Staubli VAL3: SYNCMOVE.pgx

public program syncMove(num& x_nAxisNum[])
  local jointRx l_jCurr
  local num l_nEncRes
  local num l_nDrvPos[2]
  local bool l_bFirstRun
  local num l_i
  local bool l_bError
  local string l_sMsg
begin

  l_nEncRes=8192/360

  call setCmdPos(0)
  call setCmdPos(1)
  bStop=false
  l_bFirstRun=true

  // Ne pas supprimer ces lignes
  disablePower()
  wait(isPowered()==false)
  //wait(isPowered()==true)
  /// FIN /////////////

  while !bStop
    if (isPowered()==true) and (l_bFirstRun==false)
      for l_i=0 to size(x_nAxisNum)-1
        if (diSwitchedOn[x_nAxisNum[l_i]]==false)
          doSwitchOn[x_nAxisNum[l_i]]=true
          delay(0.05)
          doEnableOp[x_nAxisNum[l_i]]=true
        endIf
      endFor
      // Get system position
      $XgetDrvCmdPos(l_nDrvPos)
      //$XgetJntCmdPos(l_nJntPos)
      // Send it to the external axis
      aioSet(aoPosCmd[x_nAxisNum[0]],l_nDrvPos[0]*l_nEncRes)
      aioSet(aoPosCmd[x_nAxisNum[1]],l_nDrvPos[1]*l_nEncRes)
      //l_sMsg="0: "+toString(".3",l_nJntPos[0])+"   1: "+toString(".3",l_nJntPos[1])
      l_sMsg="0: "+toString(".3",l_nDrvPos[0])+"   1: "+toString(".3",l_nDrvPos[1])
      //? l_sMsg
    else
      for l_i=0 to size(x_nAxisNum)-1
        doSwitchOn[x_nAxisNum[l_i]]=false
        doEnableOp[x_nAxisNum[l_i]]=false
      endFor
      // Get external axis position
      l_nDrvPos[0]=aioGet(aiPosFbk[x_nAxisNum[0]])/l_nEncRes
      l_nDrvPos[1]=aioGet(aiPosFbk[x_nAxisNum[1]])/l_nEncRes
      // Update it in the system
      $XsetDrvFbkPos(l_nDrvPos)
    endIf
    delay(0)
    l_bFirstRun=false
  endWhile
end
